# EPICS substitutions: iocBoot/iocLinux/fb_epid.substitutions
# $Id$

file "$(OPTICS)/opticsApp/Db/fb_epid.db"
  {
    {
        P=poka:epid1,
	IN=poka:epid1:sim.VAL,
	OUT=poka:epid1:sim.D,
	MODE=PID,
	CALC=A,
	PERMIT1="poka:epid1:on.VAL",
	PERMIT2="",
	PERMIT3="",
	PERMIT4=""
    }
  }
